Yaskawa INFORM job: TWIN_FRONT_SEARCH_0ST-2_5340.JBI

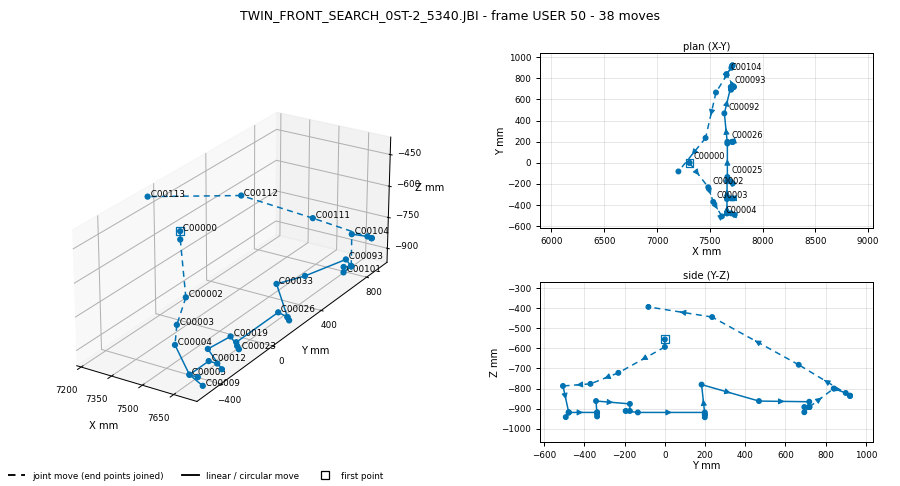
[picture p0: tool path of TWIN_FRONT_SEARCH_0ST-2_5340.JBI in frame USER 50, 38 of 42 moves have a stored position in this frame; points joined in program order, loops and branches not executed]
/JOB
//NAME TWIN_FRONT_SEARCH_0ST-2_5340
///FOLDERNAME 02-SKRZYNIE_JOBS
//POS
///NPOS 114,114,0,15,0,0
///USER 50
///TOOL 0
///POSTYPE USER
///RECTAN
///RCONF 1,0,1,0,0,0,0,0,0,0,0,0,0,0,0,0,0,0,0,0,0,0,0,0
C00000=7307.436,0.297,-555.341,-0.0028,-3.2849,0.0046
C00001=7307.427,0.296,-592.946,-0.0034,-3.2838,0.0056
///RCONF 0,0,0,0,0,0,0,0,0,0,0,0,0,0,0,0,0,0,0,0,0,0,0,0
C00002=7485.598,-231.251,-721.887,-10.9114,-20.6036,-4.2484
C00003=7532.667,-369.884,-776.575,-10.1071,-30.2492,-2.0817
C00004=7614.362,-506.862,-787.157,0.0023,-33.0550,-3.6294
C00005=7662.521,-478.139,-918.832,-3.1613,-41.6270,-1.9266
C00006=7701.887,-478.135,-918.824,-3.1611,-41.6274,-1.9267
C00007=7701.874,-478.100,-947.794,-3.1595,-41.6257,-1.9258
C00008=7753.636,-478.076,-944.774,-3.1580,-41.6265,-1.9263
C00009=7734.835,-492.833,-942.065,-45.0086,-34.6798,24.7014
C00010=7734.829,-513.428,-942.068,-45.0120,-34.6764,24.7051
C00011=7662.521,-478.139,-918.832,-3.1613,-41.6270,-1.9266
C00012=7662.802,-336.994,-918.878,-3.1595,-41.6273,-1.9277
C00013=7703.595,-336.997,-918.886,-3.1586,-41.6266,-1.9290
C00014=7703.585,-337.040,-945.410,-3.1687,-41.6262,-1.9203
C00015=7754.275,-337.021,-938.825,-3.1678,-41.6275,-1.9194
C00016=7725.540,-337.013,-938.788,36.9814,-33.0426,-26.9781
C00017=7726.047,-292.830,-938.734,53.0962,-24.5309,-34.8011
C00018=7662.513,-342.280,-862.050,-3.1593,-41.6259,-1.9277
C00019=7664.160,-173.874,-876.343,-3.1613,-41.6260,-1.9252
C00020=7695.842,-173.884,-911.532,-3.1647,-41.6259,-1.9226
C00021=7695.817,-173.881,-944.757,-3.1685,-41.6225,-1.9193
C00022=7756.799,-173.909,-941.788,-3.1728,-41.6204,-1.9170
C00023=7717.105,-194.831,-911.567,-49.6696,-32.7903,27.2913
C00024=7717.091,-227.483,-911.598,-58.6618,-27.8614,31.8083
C00025=7666.521,-134.092,-918.844,-3.1580,-41.6256,-1.9268
C00026=7666.507,198.949,-918.845,-3.1625,-41.6261,-1.9230
C00027=7712.097,198.969,-929.737,-3.1596,-41.6256,-1.9248
C00028=7712.097,198.981,-943.079,-3.1589,-41.6253,-1.9246
C00029=7756.411,198.984,-940.053,-3.1600,-41.6259,-1.9225
C00030=7720.173,198.985,-942.708,49.7429,-26.5754,-33.3515
C00031=7720.168,237.981,-942.706,49.7424,-26.5769,-33.3491
C00032=7712.097,198.969,-929.737,-3.1596,-41.6256,-1.9248
C00033=7666.512,182.875,-780.292,-3.1585,-41.6247,-1.9260
C00034=7662.521,-478.139,-918.832,-3.1613,-41.6270,-1.9266
C00035=7567.949,-506.880,-787.168,0.0025,-33.0547,-3.6304
C00036=7673.595,-531.747,-890.602,40.9162,-15.7359,-51.4312
C00037=7713.525,-520.420,-915.661,42.4213,-16.8813,-30.0823
C00038=7722.080,-517.298,-915.705,42.3866,-16.9163,-30.0492
C00039=7722.085,-503.068,-915.700,42.3871,-16.9163,-30.0497
C00040=7722.080,-517.298,-915.705,42.3866,-16.9163,-30.0492
C00041=7722.077,-517.311,-915.705,47.3530,-24.6758,-31.8178
C00042=7737.188,-517.312,-915.690,47.3540,-24.6756,-31.8197
C00043=7722.077,-517.311,-915.705,47.3530,-24.6758,-31.8178
C00044=7656.965,-517.295,-915.691,35.9692,-5.7261,-28.7820
C00045=7656.965,-517.295,-915.691,35.9692,-5.7261,-28.7820
C00046=7656.971,-490.405,-915.682,35.9681,-5.7273,-28.7800
C00047=7656.972,-490.388,-942.283,35.9685,-5.7279,-28.7791
C00048=7656.972,-490.375,-918.757,35.9689,-5.7270,-28.7788
C00049=7676.569,-751.478,-862.036,34.9694,-13.6789,-62.1832
C00050=7720.775,-743.210,-886.052,38.6770,-25.6813,-64.1276
C00051=7720.755,-751.551,-908.963,38.6789,-25.6792,-64.1311
C00052=7720.775,-743.210,-886.052,38.6770,-25.6813,-64.1276
C00053=7741.516,-743.199,-886.045,38.6809,-25.6796,-64.1295
C00054=7720.775,-743.210,-886.052,38.6770,-25.6813,-64.1276
C00055=7689.700,-926.556,-824.015,42.8653,-17.8393,-85.8488
C00056=7724.919,-926.539,-850.402,42.8639,-17.8411,-85.8463
C00057=7743.276,-926.534,-850.404,42.8657,-17.8389,-85.8479
C00058=7724.919,-926.539,-850.402,42.8639,-17.8411,-85.8463
C00059=7724.853,-926.607,-872.234,42.8635,-17.8390,-85.8512
C00060=7656.912,-926.561,-808.796,42.8626,-17.8430,-85.8460
C00061=7662.624,-440.466,-849.453,-10.3723,-28.3247,2.1721
C00062=7655.020,-61.910,-811.326,-48.3204,-9.0917,69.5388
C00063=7719.007,-0.341,-796.634,-50.3541,-9.8325,69.8718
C00064=7740.889,-0.322,-817.215,-50.3572,-9.8330,69.8742
C00065=7762.756,-0.327,-817.207,-50.3578,-9.8322,69.8744
C00066=7760.695,-0.319,-817.207,-50.3571,-9.8337,69.8740
C00067=7760.688,-0.326,-844.885,-50.3559,-9.8341,69.8727
C00068=7735.584,-0.342,-814.862,-50.3529,-9.8343,69.8702
C00069=7685.821,-442.273,-813.109,-50.3533,-9.8305,69.8722
C00070=7722.951,-442.273,-844.486,-50.3530,-9.8317,69.8712
C00071=7737.782,-442.267,-844.485,-50.3532,-9.8303,69.8722
C00072=7735.910,-442.268,-844.484,-50.3535,-9.8303,69.8723
C00073=7735.735,-442.274,-877.330,-50.3532,-9.8324,69.8704
C00074=7715.654,-442.286,-821.545,-50.3531,-9.8308,69.8708
C00075=7675.965,395.606,-804.112,-50.3525,-9.8307,69.8684
C00076=7723.190,405.651,-849.200,-50.3562,-9.8291,69.8688
C00077=7737.765,405.636,-849.214,-50.3535,-9.8303,69.8658
C00078=7735.842,405.634,-849.218,-50.3539,-9.8287,69.8668
C00079=7735.842,405.634,-874.569,-50.3542,-9.8284,69.8674
C00080=7708.320,405.630,-832.213,-50.3531,-9.8304,69.8652
C00081=7674.316,527.666,-792.803,-42.4006,-6.8574,47.1116
C00082=7727.103,501.293,-922.412,-42.3956,-6.8637,34.4317
C00083=7727.088,485.728,-922.442,-42.3934,-6.8649,34.4271
C00084=7722.614,501.285,-918.263,-42.3957,-6.8634,34.4310
C00085=7722.616,501.275,-918.253,-47.0694,-13.0045,35.2188
C00086=7736.369,501.284,-918.256,-47.0704,-13.0034,35.2202
C00087=7722.616,501.275,-918.253,-47.0694,-13.0045,35.2188
C00088=7673.748,501.298,-918.246,-30.5842,-3.3920,33.3299
C00089=7668.003,468.499,-919.193,-30.5848,-3.3919,33.3318
C00090=7667.971,468.513,-938.811,-30.5832,-3.3904,33.3312
C00091=7668.003,468.499,-919.193,-30.5848,-3.3919,33.3318
C00092=7638.065,468.471,-862.303,-30.5853,-3.3931,33.3301
C00093=7698.605,718.766,-865.669,-40.8606,-9.2184,81.3407
C00094=7725.959,718.765,-891.903,-40.8612,-9.2179,81.3427
C00095=7725.950,725.996,-910.161,-40.8620,-9.2182,81.3445
C00096=7725.959,718.765,-891.903,-40.8612,-9.2179,81.3427
C00097=7744.002,718.745,-891.885,-40.8616,-9.2181,81.3421
C00098=7725.959,718.765,-891.903,-40.8612,-9.2179,81.3427
C00099=7701.811,694.126,-891.907,-40.8628,-9.2167,81.3432
C00100=7701.844,694.095,-920.324,-40.8645,-9.2169,81.3410
C00101=7701.820,694.094,-917.813,-44.5820,14.2675,81.2031
C00102=7701.831,675.272,-917.812,-44.5827,14.2661,81.2021
C00103=7725.959,718.765,-891.903,-40.8612,-9.2179,81.3427
C00104=7658.142,840.513,-799.703,-44.7562,-8.1963,88.0277
C00105=7704.585,900.322,-822.076,-46.8259,-7.8769,99.0282
C00106=7714.362,921.598,-835.980,-46.8282,-7.8747,99.0300
C00107=7745.059,921.594,-835.961,-46.8292,-7.8744,99.0319
C00108=7714.362,921.598,-835.980,-46.8282,-7.8747,99.0300
C00109=7714.351,921.594,-872.628,-46.8270,-7.8752,99.0295
C00110=7714.362,921.598,-835.980,-46.8282,-7.8747,99.0300
C00111=7558.683,666.332,-681.732,-44.9142,-16.4186,77.8535
C00112=7459.985,235.489,-444.256,-37.0048,-34.2400,42.3881
C00113=7202.927,-81.612,-393.778,-63.8439,-12.2109,50.7232
BC00000=5880.290
BC00001=6140.111
BC00002=6140.111
BC00003=6140.111
BC00004=6140.111
BC00005=6240.111
BC00006=6240.111
BC00007=6240.111
BC00008=6240.111
BC00009=6240.111
BC00010=6240.111
BC00011=6240.111
BC00012=6240.111
BC00013=6240.111
BC00014=6240.111
BC00015=6240.111
BC00016=6240.111
BC00017=6240.111
BC00018=6240.111
BC00019=6240.111
BC00020=6240.111
BC00021=6240.118
BC00022=6240.118
BC00023=6240.111
BC00024=6240.111
BC00025=6240.111
BC00026=6240.111
BC00027=6240.111
BC00028=6240.111
BC00029=6240.111
BC00030=6240.111
BC00031=6240.111
BC00032=6240.111
BC00033=6240.111
BC00034=6240.111
BC00035=6240.111
BC00036=6240.111
BC00037=6240.111
BC00038=6240.124
BC00039=6240.124
BC00040=6240.124
BC00041=6240.124
BC00042=6240.124
BC00043=6240.124
BC00044=6240.124
BC00045=6240.124
BC00046=6240.124
BC00047=6240.124
BC00048=6240.124
BC00049=6240.124
BC00050=6240.124
BC00051=6240.124
BC00052=6240.124
BC00053=6240.124
BC00054=6240.124
BC00055=6240.124
BC00056=6240.124
BC00057=6240.124
BC00058=6240.124
BC00059=6240.124
BC00060=6240.124
BC00061=6240.131
BC00062=6240.137
BC00063=6240.137
BC00064=6240.137
BC00065=6240.137
BC00066=6240.137
BC00067=6240.137
BC00068=6240.137
BC00069=6240.137
BC00070=6240.137
BC00071=6240.137
BC00072=6240.137
BC00073=6239.955
BC00074=6240.046
BC00075=6240.046
BC00076=6240.046
BC00077=6240.046
BC00078=6240.046
BC00079=6240.046
BC00080=6240.046
BC00081=6240.137
BC00082=6240.137
BC00083=6240.137
BC00084=6240.137
BC00085=6240.137
BC00086=6240.137
BC00087=6240.137
BC00088=6240.137
BC00089=6240.137
BC00090=6240.137
BC00091=6240.137
BC00092=6240.137
BC00093=6240.137
BC00094=6240.137
BC00095=6240.137
BC00096=6240.137
BC00097=6240.137
BC00098=6240.137
BC00099=6240.137
BC00100=6240.137
BC00101=6240.137
BC00102=6240.137
BC00103=6240.137
BC00104=6240.137
BC00105=6240.137
BC00106=6240.137
BC00107=6240.137
BC00108=6240.137
BC00109=6240.137
BC00110=6240.137
BC00111=6033.217
BC00112=5861.059
BC00113=5556.515
///POSTYPE BASE
P00006=-2.449,0.031,8.825,0.0000,0.0000,0.0000
P00058=0.000,0.000,3.000,0.0000,0.0000,0.0000
P00350=11.519,-0.008,1.149,0.0000,0.0000,0.0000
P00351=13.563,-0.027,-0.653,0.0000,0.0000,0.0000
P00352=13.252,-0.027,-0.827,0.0000,0.0000,0.0000
P00353=10.971,-0.082,0.776,0.0000,0.0000,0.0000
P00399=-2.449,0.031,8.825,0.0000,0.0000,0.0000
P00400=5.920,-3.503,-0.024,0.0000,0.0000,0.0000
P00401=3.430,-0.021,1.131,0.0000,0.0000,0.0000
P00402=-0.253,1.107,3.062,0.0000,0.0000,0.0000
P00403=-3.666,-0.015,5.328,0.0000,0.0000,0.0000
P00405=2.420,0.007,1.427,0.0000,0.0000,0.0000
P00406=3.513,-0.022,0.429,0.0000,0.0000,0.0000
P00415=-1.781,-1.303,3.250,0.0000,0.0000,0.0000
P00416=0.027,1.119,3.078,0.0000,0.0000,0.0000
//INST
///DATE 2024/12/19 09:52
///ATTR SC,RW,RJ
////FRAME USER 50
///GROUP1 RB1,BS1
NOP
MOVJ C00000 BC00000 VJ=30.00
MOVJ C00001 BC00001 VJ=20.00
MOVJ C00002 BC00002 VJ=20.00
MOVJ C00003 BC00003 VJ=20.00
MOVJ C00004 BC00004 VJ=10.00
'DODANE
'SZUKANIE FRONT
'------------------------
'503
'------------------------
MOVL C00005 BC00005 V=166.7
MOVL C00006 BC00006 V=66.7 PL=0
REFP 3 C00007 BC00007
CALL JOB:SEARCH-R1
IMOV P0058 V=16.7
SET P0350 P0006
SFTON P0350
REFP 3 C00008 BC00008
CALL JOB:SEARCH-R1
SET P0350 P0006
SFTON P0350
MOVL C00009 BC00009 V=166.7
REFP 3 C00010 BC00010
CALL JOB:SEARCH-R1
SET P0350 P0006
SFTON P0350
MOVL C00011 BC00011 V=66.7 PL=0
SFTOF
'------------------------
'------------------------
'502
'------------------------
MOVL C00012 BC00012 V=166.7
MOVL C00013 BC00013 V=66.7 PL=0
REFP 3 C00014 BC00014
CALL JOB:SEARCH-R1
IMOV P0058 V=16.7
SET P0351 P0006
SFTON P0351
REFP 3 C00015 BC00015
CALL JOB:SEARCH-R1
SET P0351 P0006
SFTON P0351
MOVL C00016 BC00016 V=166.7
REFP 3 C00017 BC00017
CALL JOB:SEARCH-R1
SET P0351 P0006
SFTON P0351
MOVL C00018 BC00018 V=66.7 PL=0
SFTOF
'------------------------
'------------------------
'501
'------------------------
MOVL C00019 BC00019 V=166.7
MOVL C00020 BC00020 V=66.7 PL=0
REFP 3 C00021 BC00021
CALL JOB:SEARCH-R1
IMOV P0058 V=16.7
SET P0352 P0006
SFTON P0352
REFP 3 C00022 BC00022
CALL JOB:SEARCH-R1
SET P0352 P0006
SFTON P0352
MOVL C00023 BC00023 V=166.7
REFP 3 C00024 BC00024
CALL JOB:SEARCH-R1
SET P0352 P0006
SFTON P0352
MOVL C00025 BC00025 V=66.7 PL=0
SFTOF
'------------------------
'------------------------
'500
'------------------------
MOVL C00026 BC00026 V=166.7
MOVL C00027 BC00027 V=66.7 PL=0
REFP 3 C00028 BC00028
CALL JOB:SEARCH-R1
IMOV P0058 V=16.7
SET P0353 P0006
SFTON P0353
REFP 3 C00029 BC00029
CALL JOB:SEARCH-R1
SET P0353 P0006
SFTON P0353
MOVL C00030 BC00030 V=166.7
REFP 3 C00031 BC00031
CALL JOB:SEARCH-R1
SET P0353 P0006
SFTON P0353
MOVL C00032 BC00032 V=66.7 PL=0
SFTOF
'------------------------
MOVL C00033 BC00033 V=333.3
COMM PAUSE
COMM MOVL C00034 BC00034 V=333.3
COMM MOVJ C00035 BC00035 VJ=10.00
COMM 'DODANE
COMM MOVJ C00036 BC00036 VJ=10.00
COMM '------------------------
COMM 'SFT402
COMM '------------------------
COMM SFTOF
COMM MOVL C00037 BC00037 V=150.0
COMM MOVL C00038 BC00038 V=66.7 PL=0
COMM REFP 3 C00039 BC00039
COMM CALL JOB:SEARCH-R1
COMM SET P0402 P0006
COMM SFTON P0402
COMM MOVL C00040 BC00040 V=150.0
COMM MOVL C00041 BC00041 V=66.7 PL=0
COMM REFP 3 C00042 BC00042
COMM CALL JOB:SEARCH-R1
COMM SET P0402 P0006
COMM SFTON P0402
COMM MOVL C00043 BC00043 V=133.3
COMM MOVL C00044 BC00044 V=150.0
COMM MOVL C00045 BC00045 V=150.0
COMM MOVL C00046 BC00046 V=66.7 PL=0
COMM REFP 3 C00047 BC00047
COMM CALL JOB:SEARCH-R1
COMM SET P0402 P0006
COMM SFTOF
COMM MOVL C00048 BC00048 V=150.0
COMM '------------------------
COMM 'SFT403
COMM '------------------------
COMM 'START
COMM SFTOF
COMM MOVL C00049 BC00049 V=250.0
COMM MOVL C00050 BC00050 V=133.3 PL=0
COMM REFP 3 C00051 BC00051
COMM CALL JOB:SEARCH-R1
COMM SET P0416 P0006
COMM SFTON P0416
COMM MOVL C00052 BC00052 V=133.3
COMM REFP 3 C00053 BC00053
COMM CALL JOB:SEARCH-R1
COMM SET P0416 P0006
COMM SFTOF
COMM MOVL C00054 BC00054 V=150.0
COMM '------------------------
COMM '------------------------
COMM SFTOF
COMM MOVL C00055 BC00055 V=250.0
COMM MOVL C00056 BC00056 V=133.3 PL=0
COMM REFP 3 C00057 BC00057
COMM CALL JOB:SEARCH-R1
COMM SET P0403 P0006
COMM SFTON P0403
COMM MOVL C00058 BC00058 V=66.7 PL=0
COMM REFP 3 C00059 BC00059
COMM CALL JOB:SEARCH-R1
COMM SET P0403 P0006
COMM SFTOF
COMM MOVL C00060 BC00060 V=150.0
COMM MOVJ C00061 BC00061 VJ=20.00
COMM MOVJ C00062 BC00062 VJ=20.00
COMM '------------------------
COMM 'SFT401
COMM '------------------------
COMM SFTOF
COMM MOVL C00063 BC00063 V=150.0
COMM MOVL C00064 BC00064 V=66.7 PL=0
COMM REFP 3 C00065 BC00065
COMM CALL JOB:SEARCH-R1
COMM SET P0401 P0006
COMM SFTON P0401
COMM MOVL C00066 BC00066 V=66.7 PL=0
COMM REFP 3 C00067 BC00067
COMM CALL JOB:SEARCH-R1
COMM SET P0401 P0006
COMM SFTOF
COMM MOVL C00068 BC00068 V=150.0
COMM 'SFT400
COMM '------------------------
COMM SFTOF
COMM MOVL C00069 BC00069 V=333.3
COMM MOVL C00070 BC00070 V=66.7 PL=0
COMM REFP 3 C00071 BC00071
COMM CALL JOB:SEARCH-R1
COMM SET P0405 P0006
COMM SFTON P0405
COMM MOVL C00072 BC00072 V=66.7 PL=0
COMM REFP 3 C00073 BC00073
COMM CALL JOB:SEARCH-R1
COMM SET P0405 P0006
COMM SFTOF
COMM MOVL C00074 BC00074 V=150.0
COMM 'SFT400
COMM '------------------------
COMM SFTOF
COMM MOVL C00075 BC00075 V=333.3
COMM MOVL C00076 BC00076 V=133.3 PL=0
COMM REFP 3 C00077 BC00077
COMM CALL JOB:SEARCH-R1
COMM SET P0406 P0006
COMM SFTON P0406
COMM MOVL C00078 BC00078 V=66.7 PL=0
COMM REFP 3 C00079 BC00079
COMM CALL JOB:SEARCH-R1
COMM SET P0406 P0006
COMM SFTOF
COMM MOVL C00080 BC00080 V=150.0
COMM 'SFT400
COMM '------------------------
COMM SFTOF
COMM MOVL C00081 BC00081 V=150.0
COMM MOVL C00082 BC00082 V=66.7 PL=0
COMM REFP 3 C00083 BC00083
COMM CALL JOB:SEARCH-R1
COMM SET P0400 P0006
COMM SFTON P0400
COMM MOVL C00084 BC00084 V=150.0
COMM MOVL C00085 BC00085 V=66.7 PL=0
COMM REFP 3 C00086 BC00086
COMM CALL JOB:SEARCH-R1
COMM SET P0400 P0006
COMM SFTON P0400
COMM MOVL C00087 BC00087 V=150.0
COMM MOVL C00088 BC00088 V=150.0
COMM MOVL C00089 BC00089 V=66.7 PL=0
COMM REFP 3 C00090 BC00090
COMM CALL JOB:SEARCH-R1
COMM SET P0400 P0006
COMM SFTOF
COMM MOVL C00091 BC00091 V=83.3
COMM PAUSE
MOVL C00092 BC00092 V=250.0
MOVL C00093 BC00093 V=333.3
MOVL C00094 BC00094 V=66.7 PL=0
REFP 3 C00095 BC00095
CALL JOB:SEARCH-R1
SET P0415 P0006
SFTON P0415
MOVL C00096 BC00096 V=133.3
REFP 3 C00097 BC00097
CALL JOB:SEARCH-R1
SET P0415 P0006
SFTOF
MOVL C00098 BC00098 V=150.0
MOVL C00099 BC00099 V=66.7 PL=0
REFP 3 C00100 BC00100
CALL JOB:SEARCH-R1
SET P0416 P0006
SFTON P0416
MOVL C00101 BC00101 V=133.3
REFP 3 C00102 BC00102
CALL JOB:SEARCH-R1
SET P0416 P0006
SFTOF
MOVL C00103 BC00103 V=150.0
'------------------------
'SFT403
'------------------------
'START
SFTOF
MOVJ C00104 BC00104 VJ=10.00
'------------------------
'SFT399
'------------------------
'START
SFTOF
MOVL C00105 BC00105 V=150.0
MOVL C00106 BC00106 V=66.7 PL=0
REFP 3 C00107 BC00107
CALL JOB:SEARCH-R1
SET P0399 P0006
SFTON P0399
MOVL C00108 BC00108 V=66.7 PL=0
REFP 3 C00109 BC00109
CALL JOB:SEARCH-R1
SET P0399 P0006
SFTOF
MOVL C00110 BC00110 V=150.0
MOVJ C00111 BC00111 VJ=20.00
MOVJ C00112 BC00112 VJ=30.00
MOVJ C00113 BC00113 VJ=30.00
END
